(* IEC 61131-3 sources: CS_4_Aufzugsteuerung/src/Stations/CP112/Steuerung/Class/clsHauptablauf, 1 file *)

(* ---- clsHauptablauf.st ---- *)
(*!
<Class
	Name               = "clsHauptablauf"
	Revision           = "0.0"
	RealtimeTask       = "false"
	CyclicTask         = "true"
	DefCyclictime      = "1 ms"
	BackgroundTask     = "false"
	Sigmatek           = "false"
	OSInterface        = "false"
	HighPriority       = "false"
	Automatic          = "false"
	UpdateMode         = "Prescan"
	SharedCommandTable = "true"
	Objectsize         = "(284,120)">
	<Channels>
		<Server Name="ClassSvr" Visualized="false" Initialize="false" WriteProtected="true" Retentive="false"/>
		<Server Name="sAnf0" Visualized="true" Initialize="false" WriteProtected="true" Retentive="false"/>
		<Server Name="sAnf1" Visualized="true" Initialize="false" WriteProtected="true" Retentive="false"/>
		<Server Name="sAnf2" Visualized="true" Initialize="false" WriteProtected="true" Retentive="false"/>
		<Server Name="sAnf3" Visualized="true" Initialize="false" WriteProtected="true" Retentive="false"/>
		<Server Name="sLichtschranke" Visualized="true" Initialize="false" WriteProtected="false" Retentive="false"/>
		<Server Name="sZielEtage" Visualized="true" Initialize="false" WriteProtected="true" Retentive="false"/>
		<Client Name="cHMI" Required="true" Internal="false"/>
	</Channels>
</Class>
*)
clsHauptablauf : CLASS
  //Servers:
	ClassSvr 	: SvrChCmd_DINT;
	sAnf0 	: SvrCh_DINT;
	sAnf1 	: SvrCh_DINT;
	sAnf2 	: SvrCh_DINT;
	sAnf3 	: SvrCh_DINT;
	sLichtschranke 	: SvrCh_DINT;
	sZielEtage 	: SvrCh_DINT;
  //Clients:
	cHMI 	: CltChCmd_clsHMI;
  //Variables:
		xAnf0 	: BOOL;
		xAnf1 	: BOOL;
		xAnf2 	: BOOL;
		xAnf3 	: BOOL;
  //Functions:

	FUNCTION VIRTUAL GLOBAL CyWork
		VAR_INPUT
			EAX 	: UDINT;
		END_VAR
		VAR_OUTPUT
			state (EAX) 	: UDINT;
		END_VAR;

	FUNCTION GLOBAL Anf0
		VAR_INPUT
			xIn 	: BOOL;
		END_VAR
		VAR_OUTPUT
			xOut 	: BOOL;
		END_VAR;

	FUNCTION GLOBAL Anf1
		VAR_INPUT
			xIn 	: BOOL;
		END_VAR
		VAR_OUTPUT
			xOut 	: BOOL;
		END_VAR;

	FUNCTION GLOBAL Anf2
		VAR_INPUT
			xIn 	: BOOL;
		END_VAR
		VAR_OUTPUT
			xOut 	: BOOL;
		END_VAR;

	FUNCTION GLOBAL Anf3
		VAR_INPUT
			xIn 	: BOOL;
		END_VAR
		VAR_OUTPUT
			xOut 	: BOOL;
		END_VAR;

	FUNCTION GLOBAL TuerZu
		VAR_OUTPUT
			xOut 	: BOOL;
		END_VAR;

	FUNCTION GLOBAL TuerAuf
		VAR_OUTPUT
			xOut 	: BOOL;
		END_VAR;
  //Tables:
	FUNCTION @STD
		VAR_OUTPUT
			ret_code	: CONFSTATES;
		END_VAR;
	FUNCTION GLOBAL TAB @CT_;
END_CLASS;

#pragma usingLtd clsHMI

FUNCTION VIRTUAL GLOBAL clsHauptablauf::CyWork
	VAR_INPUT
		EAX 	: UDINT;
	END_VAR
	VAR_OUTPUT
		state (EAX) 	: UDINT;
	END_VAR

    // Hier werden zyklische Aufgaben des Hauptablaufs ausgeführt.
    // Die Anforderungsverwaltung erfolgt direkt über die Funktionen
    // Anf0() bis Anf3().

    // Neue Anforderung von HMI übernehmen
    IF cHMI.Etage0() THEN
        xAnf0 := TRUE;
    END_IF;

    // Neue Anforderung von HMI übernehmen
    IF cHMI.Etage1() THEN
        xAnf1 := TRUE;
    END_IF;

    // Neue Anforderung von HMI übernehmen
    IF cHMI.Etage2() THEN
        xAnf2 := TRUE;
    END_IF;

     // Neue Anforderung von HMI übernehmen
    IF cHMI.Etage3() THEN
        xAnf3 := TRUE;
    END_IF;

    // Weiterleitung an HMI
    //Anfragen
    IF xAnf0 THEN
      sAnf0 := 1;
    ELSE
      sAnf0 := 0;
    END_IF;

    IF xAnf1 THEN
      sAnf1 := 1;
    ELSE
      sAnf1 := 0;
    END_IF;

    IF xAnf2 THEN
      sAnf2 := 1;
    ELSE
      sAnf2 := 0;
    END_IF;

    IF xAnf3 THEN
      sAnf3 := 1;
    ELSE
      sAnf3 := 0;
    END_IF;

    //Lichtschranke
    sLichtschranke := cHMI.Lichtschranke();

    IF xAnf0 THEN
      sZielEtage := 0;
    ELSIF xAnf1 THEN
      sZielEtage := 1;
    ELSIF xAnf2 THEN
      sZielEtage := 2;
    ELSIF xAnf3 THEN
      sZielEtage := 3;
    ELSE
    sZielEtage := -1; // keine Ziel-Etage
    END_IF;

	state := READY;

END_FUNCTION

FUNCTION GLOBAL clsHauptablauf::TuerZu
	VAR_OUTPUT
		xOut 	: BOOL;
	END_VAR

  //Weitergabe von IO
   xOut := cHMI.Tuerzu();
END_FUNCTION

FUNCTION GLOBAL clsHauptablauf::TuerAuf
	VAR_OUTPUT
		xOut 	: BOOL;
	END_VAR

  //Weitergabe von IO
  IF cHMI.Tuerauf() OR (sLichtschranke <> 1) THEN //Lichtschranke MUSS 1 sein
    xOut := TRUE;
  ELSE
    xOut := FALSE;
  END_IF;

END_FUNCTION

FUNCTION GLOBAL clsHauptablauf::Anf0
	VAR_INPUT
		xIn : BOOL;          // TRUE = Anforderung zurücksetzen
	END_VAR
	VAR_OUTPUT
		xOut : BOOL;
	END_VAR

    // Anforderung löschen (z.B. nach Bedienung der Etage)
    IF xIn THEN
        xAnf0 := FALSE;
    END_IF;

    // Aktuellen Status zurückgeben
    xOut := xAnf0;

END_FUNCTION

FUNCTION GLOBAL clsHauptablauf::Anf1
	VAR_INPUT
		xIn : BOOL;
	END_VAR
	VAR_OUTPUT
		xOut : BOOL;
	END_VAR

    // Anforderung löschen
    IF xIn THEN
        xAnf1 := FALSE;
    END_IF;

    // Aktuellen Status zurückgeben
    xOut := xAnf1;

END_FUNCTION

FUNCTION GLOBAL clsHauptablauf::Anf2
	VAR_INPUT
		xIn : BOOL;
	END_VAR
	VAR_OUTPUT
		xOut : BOOL;
	END_VAR

    // Anforderung löschen
    IF xIn THEN
        xAnf2 := FALSE;
    END_IF;

    // Aktuellen Status zurückgeben
    xOut := xAnf2;

END_FUNCTION

FUNCTION GLOBAL clsHauptablauf::Anf3
	VAR_INPUT
		xIn : BOOL;
	END_VAR
	VAR_OUTPUT
		xOut : BOOL;
	END_VAR

    // Anforderung löschen
    IF xIn THEN
        xAnf3 := FALSE;
    END_IF;

    // Aktuellen Status zurückgeben
    xOut := xAnf3;

  sLichtschranke := 1;

END_FUNCTION
